FUNCTION func_f2: DINT
VAR_INPUT
    farg2_f2_x: DINT;
END_VAR
VAR
    farg_f2_x: DINT;
END_VAR


        farg_f2_x := farg2_f2_x;
IF ((farg_f2_x) <= (0)) THEN
    func_f2 := farg_f2_x;
    RETURN;
END_IF;
farg_f2_x := (farg_f2_x) - (2);
func_f2 := func_f1(farg_f2_x);
RETURN;

END_FUNCTION

(* stored: ProductVersion 3.1.0.18, Version 1.1.0.1 *)
